Yaskawa INFORM job: ILOVEYOU.JBI

/JOB
//NAME ILOVEYOU
//POS
///NPOS 58,58,58,0,0,0
///TOOL 0
///POSTYPE PULSE
///PULSE
C00000=-1523,-159448,-129981,-896,78319,82996
C00001=-53581,-4960,-56014,-65580,48677,68317
C00002=-75959,14380,-39615,-57103,41959,58059
C00003=-75828,18392,-37706,-53515,45488,60372
C00004=-75828,13522,-33771,-57703,42616,63000
C00005=-75330,11804,-35382,-57978,42943,63058
C00006=-73857,23815,-32499,-55372,46206,61042
C00007=-74089,24596,-31740,-55247,46052,61023
C00008=-74089,19923,-27891,-59288,43381,63590
C00009=-72704,25395,-22662,-60639,43932,64127
C00010=-72364,24240,-23783,-60789,44171,64147
C00011=-71182,33387,-23116,-58029,47076,62074
C00012=-71543,34383,-22095,-57859,46828,62058
C00013=-71555,34362,-22117,-57849,46823,62054
C00014=-72177,29608,-22234,-59347,45213,63185
C00015=-71568,30238,-17875,-61836,44342,64628
C00016=-70988,34587,-17246,-60616,45593,63717
C00017=-71664,34344,-22212,-57729,46794,62002
C00018=-70953,32026,-24577,-58037,47307,62016
C00019=-69780,38121,-18297,-59445,47526,62642
C00020=-70503,38889,-17424,-59048,47070,62566
C00021=-69870,37540,-10589,-63618,44965,65388
C00022=-69221,44660,-11336,-60565,47343,63242
C00023=-68900,43610,-12466,-60660,47596,63224
C00024=-67236,49685,-5852,-62527,48035,64053
C00025=-67710,51991,-3404,-62473,47617,64137
C00026=-68848,46544,-9398,-60995,47432,63437
C00027=-68848,42300,-5453,-64904,45234,65996
C00028=-67511,48826,1576,-66588,45610,66801
C00029=-67306,48123,810,-66611,45780,66774
C00030=-67306,49833,-1131,-64804,46681,65592
C00031=-67611,50221,-704,-64667,46474,65571
C00032=-68700,44814,-6588,-63252,46237,64891
C00033=-67664,41412,-10219,-63512,47057,64819
C00034=-65416,58718,3568,-64602,48528,65006
C00035=-66189,59760,5205,-64501,47871,65125
C00036=-65539,60958,11386,-67564,46885,67028
C00037=-65539,59515,13248,-69227,46143,68121
C00038=-65539,61003,11336,-67519,46906,66998
C00039=-64922,67145,13827,-66510,47945,66188
C00040=-64295,64978,11277,-66508,48508,66041
C00041=-63704,74964,22993,-68557,48018,67302
C00042=-63713,74937,22960,-68547,48015,67297
C00043=-64180,69276,21029,-69761,47073,68209
C00044=-63622,71600,27583,-72571,46436,69961
C00045=-63079,76637,29922,-71806,47167,69357
C00046=-63708,74750,22756,-68525,48030,67278
C00047=-63343,73421,21149,-68474,48373,67163
C00048=-62249,81465,31031,-70681,48323,68433
C00049=-62584,82769,32646,-70782,47998,68569
C00050=-62584,79676,37587,-74874,46504,71297
C00051=-61540,89411,49659,-77534,46560,72893
C00052=-61540,92003,44204,-73327,47874,70089
C00053=-59962,85576,36098,-72652,49430,69326
C00054=-53581,-4960,-56014,-65580,48677,68317
C00055=-1523,-159448,-129981,-896,78319,82996
C00056=-1523,-159448,-129981,-896,78319,82996
C00057=-1523,-159448,-129981,-896,78319,82996
BC00000=173457,698124,1075171
BC00001=326168,698124,386244
BC00002=326168,698124,386244
BC00003=326167,698125,386241
BC00004=326167,698125,386241
BC00005=326167,698125,386241
BC00006=326167,698125,386241
BC00007=326167,698125,386241
BC00008=326167,698125,386241
BC00009=326167,698125,386241
BC00010=326167,698125,386241
BC00011=326167,698125,386241
BC00012=326167,698125,386241
BC00013=326167,698125,386241
BC00014=326167,698125,386241
BC00015=326167,698125,386241
BC00016=326167,698125,386241
BC00017=326167,698125,386241
BC00018=326167,698125,386241
BC00019=326167,698125,386241
BC00020=326167,698125,386241
BC00021=326167,698125,386241
BC00022=326167,698125,386241
BC00023=326167,698125,386241
BC00024=326167,698125,386241
BC00025=326167,698125,386241
BC00026=326167,698125,386241
BC00027=326167,698125,386241
BC00028=326167,698125,386241
BC00029=326167,698125,386241
BC00030=326167,698125,386241
BC00031=326167,698125,386241
BC00032=326167,698125,386241
BC00033=326167,698125,386241
BC00034=326167,698125,386241
BC00035=326167,698125,386241
BC00036=326167,698125,386241
BC00037=326167,698125,386241
BC00038=326167,698125,386241
BC00039=326167,698125,386241
BC00040=326167,698125,386241
BC00041=326167,698125,386241
BC00042=326167,698125,386241
BC00043=326167,698125,386241
BC00044=326167,698125,386241
BC00045=326167,698125,386241
BC00046=326167,698125,386241
BC00047=326167,698125,386241
BC00048=326167,698125,386241
BC00049=326167,698125,386241
BC00050=326167,698125,386241
BC00051=326167,698125,386241
BC00052=326167,698125,386241
BC00053=326167,698125,386241
BC00054=326168,698124,386244
BC00055=173457,698124,1075171
BC00056=173457,698124,1075171
BC00057=173457,698124,1075171
EC00000=-4,1112950
EC00001=-4,1246897
EC00002=-4,1246897
EC00003=-5,1246896
EC00004=-5,1246896
EC00005=-5,1246896
EC00006=-5,1246896
EC00007=-5,1246896
EC00008=-5,1246896
EC00009=-5,1246896
EC00010=-5,1246896
EC00011=-5,1246896
EC00012=-5,1246896
EC00013=-5,1246896
EC00014=-5,1246896
EC00015=-5,1246896
EC00016=-5,1246896
EC00017=-5,1246896
EC00018=-5,1246896
EC00019=-5,1246896
EC00020=-5,1246896
EC00021=-5,1246896
EC00022=-5,1246896
EC00023=-5,1246896
EC00024=-5,1246896
EC00025=-5,1246896
EC00026=-5,1246896
EC00027=-5,1246896
EC00028=-5,1246896
EC00029=-5,1246896
EC00030=-5,1246896
EC00031=-5,1246896
EC00032=-5,1246896
EC00033=-5,1246896
EC00034=-5,1246896
EC00035=-5,1246896
EC00036=-5,1246896
EC00037=-5,1246896
EC00038=-5,1246896
EC00039=-5,1246896
EC00040=-5,1246896
EC00041=-5,1246896
EC00042=-5,1246896
EC00043=-5,1246896
EC00044=-5,1246896
EC00045=-5,1246896
EC00046=-5,1246896
EC00047=-5,1246896
EC00048=-5,1246896
EC00049=-5,1246896
EC00050=-5,1246896
EC00051=-5,1246896
EC00052=-5,1246896
EC00053=-5,1246896
EC00054=-4,1246897
EC00055=-4,1267313
EC00056=150635,1349057
EC00057=-4,1112950
//INST
///DATE 2024/03/24 20:37
///ATTR SC,RW
///GROUP1 RB1,BS1
///GROUP2 ST1
NOP
MOVJ C00000 BC00000 VJ=100.00  +MOVJ EC00000 VJ=100.00
MOVJ C00001 BC00001 VJ=100.00  +MOVJ EC00001 VJ=100.00
MOVJ C00002 BC00002 VJ=60.00  +MOVJ EC00002 VJ=100.00
SMOVL C00003 BC00003 V=33.3  +MOVJ EC00003
SMOVL C00004 BC00004 V=33.3  +MOVJ EC00004
SMOVL C00005 BC00005 V=33.3  +MOVJ EC00005
SMOVL C00006 BC00006 V=500.0  +MOVJ EC00006
SMOVL C00007 BC00007 V=33.3  +MOVJ EC00007
SMOVL C00008 BC00008 V=33.3  +MOVJ EC00008
SMOVL C00009 BC00009 V=33.3  +MOVJ EC00009
SMOVL C00010 BC00010 V=33.3  +MOVJ EC00010
SMOVL C00011 BC00011 V=500.0  +MOVJ EC00011
SMOVL C00012 BC00012 V=33.3  +MOVJ EC00012
SMOVC C00013 BC00013 V=33.3  +MOVJ EC00013
SMOVC C00014 BC00014 V=33.3  +MOVJ EC00014
SMOVC C00015 BC00015 V=33.3  +MOVJ EC00015
SMOVC C00016 BC00016 V=33.3  +MOVJ EC00016
SMOVC C00017 BC00017 V=33.3  +MOVJ EC00017
SMOVL C00018 BC00018 V=500.0  +MOVJ EC00018
SMOVL C00019 BC00019 V=500.0  +MOVJ EC00019
SMOVL C00020 BC00020 V=33.3  +MOVJ EC00020
SMOVL C00021 BC00021 V=33.3  +MOVJ EC00021
SMOVL C00022 BC00022 V=33.3  +MOVJ EC00022
SMOVL C00023 BC00023 V=33.3  +MOVJ EC00023
SMOVL C00024 BC00024 V=500.0  +MOVJ EC00024
SMOVL C00025 BC00025 V=33.3  +MOVJ EC00025
SMOVL C00026 BC00026 V=33.3  +MOVJ EC00026
SMOVL C00027 BC00027 V=33.3  +MOVJ EC00027
SMOVL C00028 BC00028 V=33.3  +MOVJ EC00028
SMOVL C00029 BC00029 V=33.3  +MOVJ EC00029
SMOVL C00030 BC00030 V=33.3  +MOVJ EC00030
SMOVL C00031 BC00031 V=33.3  +MOVJ EC00031
SMOVL C00032 BC00032 V=33.3  +MOVJ EC00032
SMOVL C00033 BC00033 V=33.3  +MOVJ EC00033
SMOVL C00034 BC00034 V=500.0  +MOVJ EC00034
SMOVL C00035 BC00035 V=33.3  +MOVJ EC00035
SMOVL C00036 BC00036 V=33.3  +MOVJ EC00036
SMOVL C00037 BC00037 V=33.3  +MOVJ EC00037
SMOVL C00038 BC00038 V=33.3  +MOVJ EC00038
SMOVL C00039 BC00039 V=33.3  +MOVJ EC00039
SMOVL C00040 BC00040 V=33.3  +MOVJ EC00040
SMOVL C00041 BC00041 V=33.3  +MOVJ EC00041
SMOVC C00042 BC00042 V=33.3  +MOVJ EC00042
SMOVC C00043 BC00043 V=33.3  +MOVJ EC00043
SMOVC C00044 BC00044 V=33.3  +MOVJ EC00044
SMOVC C00045 BC00045 V=33.3  +MOVJ EC00045
SMOVC C00046 BC00046 V=33.3  +MOVJ EC00046
SMOVL C00047 BC00047 V=33.3  +MOVJ EC00047
SMOVL C00048 BC00048 V=33.3  +MOVJ EC00048
SMOVL C00049 BC00049 V=33.3  +MOVJ EC00049
SMOVL C00050 BC00050 V=33.3  +MOVJ EC00050
SMOVL C00051 BC00051 V=33.3  +MOVJ EC00051
SMOVL C00052 BC00052 V=33.3  +MOVJ EC00052
SMOVL C00053 BC00053 V=250.0  +MOVJ EC00053
SMOVL C00054 BC00054 V=500.0  +MOVJ EC00054
MOVJ C00055 BC00055 VJ=100.00  +MOVJ EC00055 VJ=100.00
MOVJ C00056 BC00056 VJ=100.00  +MOVJ EC00056 VJ=100.00
TIMER T=5.00
MOVJ C00057 BC00057 VJ=100.00  +MOVJ EC00057 VJ=100.00
END
